Fanuc KAREL source: kx00018.KL

-- PROVISIONAL review KL for V940-1; original PC SHA256 4a5be4d9dc33fa235bf8340b12c91fb04f2ba74cd4024c45926c78f262e8258c
-- Incomplete behavior may be omitted. Consult companion uncertainty JSON. Do not deploy.
PROGRAM KX00018
%NOLOCKGROUP
VAR
  I : INTEGER
  J : INTEGER
  B : BOOLEAN
  F : FILE
  S : STRING[80]
-- UNRESOLVED_DECL P type=000102
-- UNRESOLVED_DECL BA type=002018
BEGIN
  -- V9_ZERO_TABLE_METADATA_HINT layout=0001; no indexed target words; source/name/runtime held
  -- UNRESOLVED_PC offsets 5-19; opcodes 2E,22,9D,33,B2
  -- UNRESOLVED_PC offsets 24-39; opcodes 22,9D,33,B1,23
  -- UNRESOLVED_PC offsets 44-48; opcodes 7F
END KX00018
